FUNCTION_BLOCK R_TRIG (* IEC 61131-3 Table 35,#1 *)
  (* Standard: 61131-3 *)
  (* Version 0.0, 2004-12-15, JHC, Rockwell Automation, Converted from SRC format. *)
  (* Compiler header: package fb.rt.plc; *)
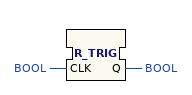
  VAR_INPUT
    CLK : BOOL;
  END_VAR
  VAR_OUTPUT
    Q : BOOL;
  END_VAR
  VAR
    M : BOOL;
  END_VAR
  ALGORITHM REQ IN ST:
Q:=CLK&NOT M;
M:=CLK;
  END_ALGORITHM
END_FUNCTION_BLOCK
